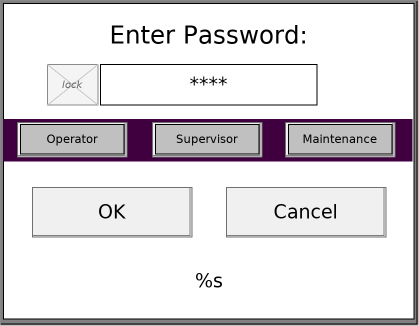
VISUALIZATION Std_Password  // 419x326
    Group (0,0 415x322)
        Rectangle (0,0 417x324)
        RoundedRectangle (3,3 411x316)
    Rectangle (3,119 409x42)
    RoundedRectangle (89,20 240x30), "Enter Password:"
    Rectangle (100,64 217x41), "****", text variable: Global_Variables_Holding.Password_Control .In_EntryPasswordString
        OnMouseDown: write the text variable via Edit, min 0, max 10, password
    Button (32,187 160x50), "OK"
        tap Global_Variables_Holding.Password_Control .In_EnterPassword
    Button (226,187 160x50), "Cancel"
        OnMouseUp: change screen: AssignExpression TP00_MAIN
    RoundedRectangle (89,266 240x30), "%s", text variable: Global_Variables_Holding.Password_Control .Out_StatusString
    Image (47,64 51x41), image: lock
    Button (17,122 110x35), "Operator"
        OnMouseUp: execute { Global_Variables_Holding.Password_Control .In_SelectedPasswordLvl:=(0); }
    Button (152,122 110x35), "Supervisor"
        OnMouseUp: execute { Global_Variables_Holding.Password_Control .In_SelectedPasswordLvl:=(1); }
    Button (285,122 110x35), "Maintenance"
        OnMouseUp: execute { Global_Variables_Holding.Password_Control .In_SelectedPasswordLvl:=(2); }
    RoundedRectangle (20,124 104x30), "Operator", colour toggle: Global_Variables_Holding.Password_Control .In_SelectedPasswordLvl = 0
        OnMouseUp: execute { Global_Variables_Holding.Password_Control .In_SelectedPasswordLvl:=(0); }
    RoundedRectangle (155,124 104x30), "Supervisor", colour toggle: Global_Variables_Holding.Password_Control .In_SelectedPasswordLvl = 1
        OnMouseUp: execute { Global_Variables_Holding.Password_Control .In_SelectedPasswordLvl:=(1); }
    RoundedRectangle (288,124 104x30), "Maintenance", colour toggle: Global_Variables_Holding.Password_Control .In_SelectedPasswordLvl = 2
        OnMouseUp: execute { Global_Variables_Holding.Password_Control .In_SelectedPasswordLvl:=(2); }
END_VISUALIZATION

(* stored: Version 1.1.0.1, ProductVersion 3.1.4018.2
   Visu Std_Password: Id {60b18236-3e1b-407f-9599-d23706fbf049} *)
